FUNCTION_BLOCK CarriageModel
  (* Standard: 61499-2 *)
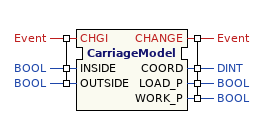
  EVENT_INPUT
    CHGI WITH INSIDE, OUTSIDE;
  END_EVENT
  EVENT_OUTPUT
    CHANGE WITH LOAD_P, WORK_P, COORD;
  END_EVENT
  VAR_INPUT
    INSIDE : BOOL;
    OUTSIDE : BOOL;
  END_VAR
  VAR_OUTPUT
    COORD : DINT;
    LOAD_P : BOOL;
    WORK_P : BOOL;
  END_VAR
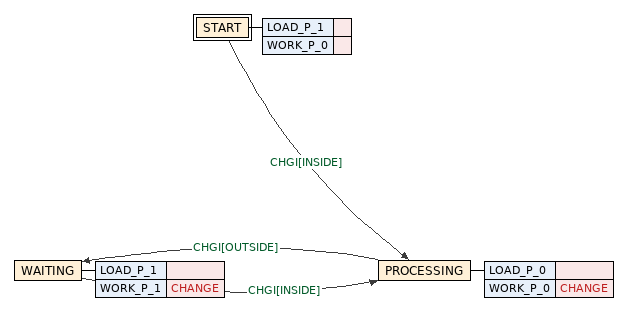
  EC_STATES
    START : LOAD_P_1, WORK_P_0;
    PROCESSING : LOAD_P_0, WORK_P_0 -> CHANGE;
    WAITING : LOAD_P_1, WORK_P_1 -> CHANGE;
  END_STATES
  EC_TRANSITIONS
    START TO PROCESSING := CHGI[INSIDE];
    PROCESSING TO WAITING := CHGI[OUTSIDE];
    WAITING TO PROCESSING := CHGI[INSIDE];
  END_TRANSITIONS
  ALGORITHM LOAD_P_0 IN ST:
LOAD_P := FALSE;&#10;
  END_ALGORITHM
  ALGORITHM LOAD_P_1 IN ST:
LOAD_P := TRUE;&#10;
  END_ALGORITHM
  ALGORITHM WORK_P_0 IN ST:
WORK_P := FALSE;&#10;
  END_ALGORITHM
  ALGORITHM WORK_P_1 IN ST:
WORK_P := TRUE;&#10;
  END_ALGORITHM
END_FUNCTION_BLOCK
